TYPE TcoKrc4_Inputs_v_5_x_x : 
STRUCT
    Inputs AT %I* : ARRAY[0..63] OF BYTE;
END_STRUCT
END_TYPE

(* stored: Version 1.1.0.1, ProductVersion 3.1.4024.12
   DUT TcoKrc4_Inputs_v_5_x_x: Id {29534d7d-068e-0c77-3675-b188d4ac803b} *)
